(*			
	RAFALOS
	Rafał Osajda		19.09.2025		TC 4024.66
	Moduł logujący wszsytkie zgłoszenia
*)
FUNCTION_BLOCK FB_Logger IMPLEMENTS ITF_Logger
VAR
END_VAR

END_FUNCTION_BLOCK

(* stored: Version 1.1.0.1
   POU FB_Logger: Id {e337bc65-3f4c-06e8-12c9-a1d49597b716}, SpecialFunc None *)
